{attribute 'qualified_only'}
{attribute 'strict'}
{attribute 'to_string'}
TYPE E_Season :
(
    Autumn,
    Winter,
    Spring,
    Summer
);
END_TYPE

(* stored: Version 1.1.0.1, ProductVersion 3.1.4024.12
   DUT E_Season: Id {0919d227-6a8b-4ea6-a538-0e150a127bd5} *)
